Fanuc KAREL source: READ_KB.kl

PROGRAM T
%NOLOCKGROUP
VAR
 v0 : FILE
 v1 : STRING[40]
 v2 : INTEGER
 v3 : INTEGER
 v4 : INTEGER
 v5 : INTEGER
 v6 : STRING[40]
 v7 : INTEGER
 v8 : INTEGER
 v9 : INTEGER
BEGIN
 READ_KB(v0, v1, v2, v3, v4, v5, v6, v7, v8, v9)
END T
